(* CODESYS project Prova_Ladder_e_ST.project

Project tree, tasks and I/O mapping:
  Device : CODESYS Control Win V3, 3S - Smart Software Solutions GmbH, order no. 305021, version 3.5.10.30
    application Application
      libraries: Standard, * (System)
      task MainTask (cyclic, interval t#20ms, priority 1) calls PLC_PRG, ST_POU
      task VISU_TASK (cyclic, interval 100 ms, priority 31) calls VisuElems.Visu_Prg
      program PLC_PRG [LD]
      visualisation Visualization
      program ST_POU [ST]
  text list GlobalTextList
*)

// Device/Application/PLC_PRG
PROGRAM PLC_PRG
VAR
	Contact1: BOOL;
	Coil1: BOOL;
END_VAR

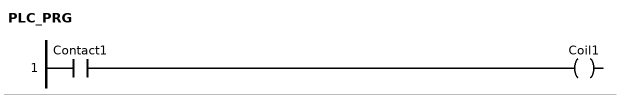
// NETWORK 1
Coil1 := Contact1;

END_PROGRAM

// Device/Application/ST_POU
PROGRAM ST_POU
VAR
	Contact1: BOOL;
	Coil1: BOOL;
END_VAR

IF Contact1 = TRUE THEN;
	Coil1 := TRUE;
ELSE
	Coil1 := FALSE;
END_IF

END_PROGRAM

// Device/Application/Visualization
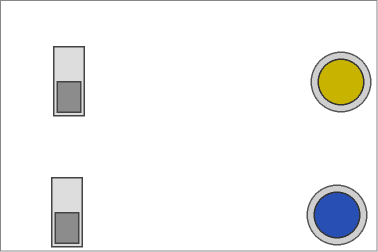
VISUALIZATION Visualization  // 378x252
    DipSwitch (34,46 70x70), variable: PLC_PRG.Contact1, behaviour: TOGGLE, style: Switch-DipSwitch-Gray
    Lamp1 (306,47 70x70), variable: PLC_PRG.Coil1, style: Lamp-Lamp1-Yellow
    Lamp1 (302,180 70x70), variable: ST_POU.Coil1, style: Lamp-Lamp1-Blue
    DipSwitch (32,177 70x70), variable: ST_POU.Contact1, behaviour: TOGGLE, style: Switch-DipSwitch-Gray
END_VISUALIZATION
